{attribute 'pack_mode' := '1'}
TYPE ST_AdsSumReadRequest :
STRUCT
	IndexGroup : UDINT;
	IndexOffset : UDINT;
	Length : UDINT;
END_STRUCT
END_TYPE

(* stored: Version 1.1.0.1, ProductVersion 3.1.4026.18
   DUT ST_AdsSumReadRequest: Id {fd38eda0-48f1-4b8a-a0b4-46f29640ccfa} *)
